(* IEC 61131-3 sources: StarkHacks-Guide-for-PLC-Troubleshooting-Tool/, 8 files *)

(* ---- codesys_constants.st ---- *)
(*
    codesys_constants.st
    Add this as a DUT or global constants list in CODESYS.
    Use these values so the PLC code, Modbus map, Python bridge, and docs all speak the same language.
*)

VAR_GLOBAL CONSTANT
    MODE_IDLE : INT := 0;
    MODE_CONVEYOR : INT := 1;
    MODE_SEQUENCE_TEST : INT := 2;
    MODE_TANK_FILL : INT := 3;
    MODE_HVAC_PUMP : INT := 4;

    FAULT_NONE : INT := 0;
    FAULT_START_BLOCKED_SAFETY : INT := 101;
    FAULT_CONVEYOR_JAM : INT := 201;
    FAULT_SEQUENCE_TIMEOUT : INT := 301;
    FAULT_TANK_FILL_VERIFY : INT := 401;
    FAULT_HVAC_OR_PUMP : INT := 501;
END_VAR

(* ---- codesys_globals.st ---- *)
(*
    codesys_globals.st
    Create a Global Variable List (GVL) in CODESYS and paste this content into it.
    These variables are the shared machine state used by all demo scenarios and the Modbus map.
*)

{attribute 'qualified_only'}
VAR_GLOBAL
    Conveyor_Running : BOOL := FALSE;      (* HR0 *)
    Sensor_Blocked : BOOL := FALSE;        (* HR1 *)
    Motor_Current : INT := 0;              (* HR2 *)
    Safety_OK : BOOL := TRUE;              (* HR3 *)
    Start_Command : BOOL := FALSE;         (* HR4 *)
    Stop_Command : BOOL := FALSE;          (* HR5 *)
    Reset_Command : BOOL := FALSE;         (* HR6 *)
    Tank_Level_Low : BOOL := FALSE;        (* HR7 *)
    Tank_Level_High : BOOL := FALSE;       (* HR8 *)
    Sequence_Timeout : BOOL := FALSE;      (* HR9 *)
    System_Fault_Latch : BOOL := FALSE;    (* HR10 *)
    Pump_Running : BOOL := FALSE;          (* HR11 *)
    HVAC_Fault : BOOL := FALSE;            (* HR12 *)
    Mode_Code : INT := 0;                  (* HR13 *)
    Fault_Code : INT := 0;                 (* HR14 *)

    Demo_EnableAutoCurrentModel : BOOL := TRUE;
    Demo_JamTimerPreset : TIME := T#3S;
    Demo_SequenceTimerPreset : TIME := T#8S;
    Demo_FillGuardPreset : TIME := T#5S;
END_VAR

(* ---- codesys_demo_supervisor.st ---- *)
(*
    codesys_demo_supervisor.st
    Optional helper block for demo stability.
    Call this once per scan to keep unrelated outputs quiet when switching modes.
*)

FUNCTION_BLOCK FB_DemoSupervisor
VAR_INPUT
    Mode_Code : INT;
    Stop_Command : BOOL;
END_VAR
VAR_IN_OUT
    Conveyor_Running : BOOL;
    Pump_Running : BOOL;
END_VAR

IF Stop_Command THEN
    Conveyor_Running := FALSE;
    Pump_Running := FALSE;
END_IF;

CASE Mode_Code OF
    MODE_CONVEYOR, MODE_SEQUENCE_TEST:
        Pump_Running := FALSE;
    MODE_TANK_FILL, MODE_HVAC_PUMP:
        Conveyor_Running := FALSE;
ELSE
    Conveyor_Running := FALSE;
    Pump_Running := FALSE;
END_CASE;

(* ---- codesys_fb_conveyor_demo.st ---- *)
(*
    codesys_fb_conveyor_demo.st
    Function block for conveyor-related demo behavior:
    - start blocked by safety
    - conveyor running logic
    - jam detection
    - sequence timeout support when Mode_Code = 2
*)

FUNCTION_BLOCK FB_ConveyorDemo
VAR_INPUT
    Safety_OK : BOOL;
    Start_Command : BOOL;
    Stop_Command : BOOL;
    Reset_Command : BOOL;
    Sensor_Blocked : BOOL;
    Mode_Code : INT;
    FaultLatchedIn : BOOL;
    JamTimerPreset : TIME;
    SequenceTimerPreset : TIME;
END_VAR
VAR_IN_OUT
    Conveyor_Running : BOOL;
    Motor_Current : INT;
    Sequence_Timeout : BOOL;
    System_Fault_Latch : BOOL;
    Fault_Code : INT;
END_VAR
VAR
    StartEdge : R_TRIG;
    ResetEdge : R_TRIG;
    JamTimer : TON;
    SequenceTimer : TON;
END_VAR

StartEdge(CLK := Start_Command);
ResetEdge(CLK := Reset_Command);

IF Stop_Command THEN
    Conveyor_Running := FALSE;
END_IF;

IF Start_Command AND NOT Safety_OK THEN
    Conveyor_Running := FALSE;
    System_Fault_Latch := TRUE;
    Fault_Code := FAULT_START_BLOCKED_SAFETY;
END_IF;

IF StartEdge.Q AND Safety_OK AND NOT FaultLatchedIn AND (Mode_Code = MODE_CONVEYOR OR Mode_Code = MODE_SEQUENCE_TEST) THEN
    Conveyor_Running := TRUE;
END_IF;

JamTimer(IN := (Mode_Code = MODE_CONVEYOR) AND Conveyor_Running AND Sensor_Blocked, PT := JamTimerPreset);
IF JamTimer.Q THEN
    Conveyor_Running := FALSE;
    System_Fault_Latch := TRUE;
    Fault_Code := FAULT_CONVEYOR_JAM;
END_IF;

SequenceTimer(IN := (Mode_Code = MODE_SEQUENCE_TEST) AND Conveyor_Running AND NOT Sensor_Blocked, PT := SequenceTimerPreset);
IF SequenceTimer.Q THEN
    Sequence_Timeout := TRUE;
    Conveyor_Running := FALSE;
    System_Fault_Latch := TRUE;
    Fault_Code := FAULT_SEQUENCE_TIMEOUT;
END_IF;

IF Conveyor_Running AND Sensor_Blocked THEN
    Motor_Current := 46;
ELSIF Conveyor_Running THEN
    Motor_Current := 18;
ELSE
    Motor_Current := 0;
END_IF;

IF ResetEdge.Q AND Safety_OK AND NOT Sensor_Blocked THEN
    IF Fault_Code = FAULT_CONVEYOR_JAM OR Fault_Code = FAULT_START_BLOCKED_SAFETY OR Fault_Code = FAULT_SEQUENCE_TIMEOUT THEN
        Conveyor_Running := FALSE;
        Sequence_Timeout := FALSE;
        IF Fault_Code <> FAULT_HVAC_OR_PUMP AND Fault_Code <> FAULT_TANK_FILL_VERIFY THEN
            System_Fault_Latch := FALSE;
            Fault_Code := FAULT_NONE;
        END_IF;
    END_IF;
END_IF;

(* ---- codesys_fb_hvac_demo.st ---- *)
(*
    codesys_fb_hvac_demo.st
    Function block for the HVAC / remote pump demo.
*)

FUNCTION_BLOCK FB_HVACDemo
VAR_INPUT
    HVAC_Fault : BOOL;
    Start_Command : BOOL;
    Stop_Command : BOOL;
    Reset_Command : BOOL;
    Mode_Code : INT;
END_VAR
VAR_IN_OUT
    Pump_Running : BOOL;
    System_Fault_Latch : BOOL;
    Fault_Code : INT;
END_VAR
VAR
    ResetEdge : R_TRIG;
END_VAR

ResetEdge(CLK := Reset_Command);

IF Mode_Code <> MODE_HVAC_PUMP THEN
    RETURN;
END_IF;

IF Stop_Command THEN
    Pump_Running := FALSE;
END_IF;

IF Start_Command AND NOT HVAC_Fault AND NOT System_Fault_Latch THEN
    Pump_Running := TRUE;
END_IF;

IF HVAC_Fault THEN
    Pump_Running := FALSE;
    System_Fault_Latch := TRUE;
    Fault_Code := FAULT_HVAC_OR_PUMP;
END_IF;

IF ResetEdge.Q AND NOT HVAC_Fault THEN
    IF Fault_Code = FAULT_HVAC_OR_PUMP THEN
        Pump_Running := FALSE;
        System_Fault_Latch := FALSE;
        Fault_Code := FAULT_NONE;
    END_IF;
END_IF;

(* ---- codesys_fb_tank_fill_demo.st ---- *)
(*
    codesys_fb_tank_fill_demo.st
    Function block for the tank fill verification demo.
*)

FUNCTION_BLOCK FB_TankFillDemo
VAR_INPUT
    Tank_Level_Low : BOOL;
    Tank_Level_High : BOOL;
    Stop_Command : BOOL;
    Reset_Command : BOOL;
    Mode_Code : INT;
    FaultLatchedIn : BOOL;
    FillGuardPreset : TIME;
END_VAR
VAR_IN_OUT
    Pump_Running : BOOL;
    System_Fault_Latch : BOOL;
    Fault_Code : INT;
END_VAR
VAR
    ResetEdge : R_TRIG;
    FillGuardTimer : TON;
END_VAR

ResetEdge(CLK := Reset_Command);

IF Mode_Code <> MODE_TANK_FILL THEN
    FillGuardTimer(IN := FALSE, PT := FillGuardPreset);
    RETURN;
END_IF;

IF Stop_Command THEN
    Pump_Running := FALSE;
END_IF;

IF Tank_Level_Low AND NOT Tank_Level_High AND NOT FaultLatchedIn THEN
    Pump_Running := TRUE;
END_IF;

IF Tank_Level_High THEN
    Pump_Running := FALSE;
END_IF;

FillGuardTimer(IN := Tank_Level_Low AND NOT Tank_Level_High AND NOT Pump_Running, PT := FillGuardPreset);
IF FillGuardTimer.Q THEN
    System_Fault_Latch := TRUE;
    Fault_Code := FAULT_TANK_FILL_VERIFY;
END_IF;

IF ResetEdge.Q AND NOT Tank_Level_Low AND NOT Tank_Level_High THEN
    IF Fault_Code = FAULT_TANK_FILL_VERIFY THEN
        Pump_Running := FALSE;
        System_Fault_Latch := FALSE;
        Fault_Code := FAULT_NONE;
    END_IF;
END_IF;

(* ---- codesys_main_program.st ---- *)
(*
    codesys_main_program.st
    Recommended main PLC program for the demo.

    This version is more modular than plc_logic.st.
    Use this if you want a cleaner CODESYS structure with separate function blocks per scenario.
*)

PROGRAM PLC_PRG
VAR
    ConveyorDemo : FB_ConveyorDemo;
    TankFillDemo : FB_TankFillDemo;
    HVACDemo : FB_HVACDemo;
    DemoSupervisor : FB_DemoSupervisor;
END_VAR

IF GVL_Diagnostics.Reset_Command THEN
    IF GVL_Diagnostics.Safety_OK AND NOT GVL_Diagnostics.Sensor_Blocked AND NOT GVL_Diagnostics.HVAC_Fault THEN
        GVL_Diagnostics.Sequence_Timeout := FALSE;
    END_IF;
END_IF;

DemoSupervisor(
    Mode_Code := GVL_Diagnostics.Mode_Code,
    Stop_Command := GVL_Diagnostics.Stop_Command,
    Conveyor_Running := GVL_Diagnostics.Conveyor_Running,
    Pump_Running := GVL_Diagnostics.Pump_Running
);

ConveyorDemo(
    Safety_OK := GVL_Diagnostics.Safety_OK,
    Start_Command := GVL_Diagnostics.Start_Command,
    Stop_Command := GVL_Diagnostics.Stop_Command,
    Reset_Command := GVL_Diagnostics.Reset_Command,
    Sensor_Blocked := GVL_Diagnostics.Sensor_Blocked,
    Mode_Code := GVL_Diagnostics.Mode_Code,
    FaultLatchedIn := GVL_Diagnostics.System_Fault_Latch,
    JamTimerPreset := GVL_Diagnostics.Demo_JamTimerPreset,
    SequenceTimerPreset := GVL_Diagnostics.Demo_SequenceTimerPreset,
    Conveyor_Running := GVL_Diagnostics.Conveyor_Running,
    Motor_Current := GVL_Diagnostics.Motor_Current,
    Sequence_Timeout := GVL_Diagnostics.Sequence_Timeout,
    System_Fault_Latch := GVL_Diagnostics.System_Fault_Latch,
    Fault_Code := GVL_Diagnostics.Fault_Code
);

TankFillDemo(
    Tank_Level_Low := GVL_Diagnostics.Tank_Level_Low,
    Tank_Level_High := GVL_Diagnostics.Tank_Level_High,
    Stop_Command := GVL_Diagnostics.Stop_Command,
    Reset_Command := GVL_Diagnostics.Reset_Command,
    Mode_Code := GVL_Diagnostics.Mode_Code,
    FaultLatchedIn := GVL_Diagnostics.System_Fault_Latch,
    FillGuardPreset := GVL_Diagnostics.Demo_FillGuardPreset,
    Pump_Running := GVL_Diagnostics.Pump_Running,
    System_Fault_Latch := GVL_Diagnostics.System_Fault_Latch,
    Fault_Code := GVL_Diagnostics.Fault_Code
);

HVACDemo(
    HVAC_Fault := GVL_Diagnostics.HVAC_Fault,
    Start_Command := GVL_Diagnostics.Start_Command,
    Stop_Command := GVL_Diagnostics.Stop_Command,
    Reset_Command := GVL_Diagnostics.Reset_Command,
    Mode_Code := GVL_Diagnostics.Mode_Code,
    Pump_Running := GVL_Diagnostics.Pump_Running,
    System_Fault_Latch := GVL_Diagnostics.System_Fault_Latch,
    Fault_Code := GVL_Diagnostics.Fault_Code
);

(* ---- plc_logic.st ---- *)
(*
    plc_logic.st
    Sample Structured Text logic for the hackathon prototype.

    Notes:
    - Map these variables to the holding registers documented in register_map.md.
    - Factory I/O should drive the simulated sensors and read the actuator outputs.
    - This is a compact demo program, not a production safety program.
*)

PROGRAM PLC_PRG
VAR
    Conveyor_Running : BOOL := FALSE;      (* HR0 *)
    Sensor_Blocked : BOOL := FALSE;        (* HR1 *)
    Motor_Current : INT := 0;              (* HR2 *)
    Safety_OK : BOOL := TRUE;              (* HR3 *)
    Start_Command : BOOL := FALSE;         (* HR4 *)
    Stop_Command : BOOL := FALSE;          (* HR5 *)
    Reset_Command : BOOL := FALSE;         (* HR6 *)
    Tank_Level_Low : BOOL := FALSE;        (* HR7 *)
    Tank_Level_High : BOOL := FALSE;       (* HR8 *)
    Sequence_Timeout : BOOL := FALSE;      (* HR9 *)
    System_Fault_Latch : BOOL := FALSE;    (* HR10 *)
    Pump_Running : BOOL := FALSE;          (* HR11 *)
    HVAC_Fault : BOOL := FALSE;            (* HR12 *)
    Mode_Code : INT := 0;                  (* HR13 *)
    Fault_Code : INT := 0;                 (* HR14 *)

    StartEdge : R_TRIG;
    ResetEdge : R_TRIG;
    JamTimer : TON;
    SequenceTimer : TON;
    FillGuardTimer : TON;
END_VAR

(* Edge detectors *)
StartEdge(CLK := Start_Command);
ResetEdge(CLK := Reset_Command);

(* Defaults *)
Sequence_Timeout := FALSE;

(* Stop command always drops outputs *)
IF Stop_Command THEN
    Conveyor_Running := FALSE;
    Pump_Running := FALSE;
END_IF;

(* Safety blocked start check *)
IF Start_Command AND NOT Safety_OK THEN
    Conveyor_Running := FALSE;
    System_Fault_Latch := TRUE;
    Fault_Code := 101;
END_IF;

(* Healthy start behavior *)
IF StartEdge.Q AND Safety_OK AND NOT System_Fault_Latch THEN
    CASE Mode_Code OF
        1: Conveyor_Running := TRUE;
        2: Conveyor_Running := TRUE;
        3: Pump_Running := Tank_Level_Low AND NOT Tank_Level_High;
        4: Pump_Running := TRUE;
    ELSE
        Conveyor_Running := FALSE;
        Pump_Running := FALSE;
    END_CASE;
END_IF;

(* Conveyor jam logic *)
JamTimer(IN := Conveyor_Running AND Sensor_Blocked, PT := T#3S);
IF JamTimer.Q THEN
    System_Fault_Latch := TRUE;
    Fault_Code := 201;
    Conveyor_Running := FALSE;
END_IF;

(* Sequence timing validation mode *)
SequenceTimer(IN := (Mode_Code = 2) AND Conveyor_Running AND NOT Tank_Level_High, PT := T#8S);
IF SequenceTimer.Q THEN
    Sequence_Timeout := TRUE;
    System_Fault_Latch := TRUE;
    Fault_Code := 301;
    Conveyor_Running := FALSE;
END_IF;

(* Tank fill verification mode *)
IF Mode_Code = 3 THEN
    IF Tank_Level_Low AND NOT System_Fault_Latch THEN
        Pump_Running := TRUE;
    END_IF;

    IF Tank_Level_High THEN
        Pump_Running := FALSE;
    END_IF;

    FillGuardTimer(IN := Tank_Level_Low AND NOT Tank_Level_High AND NOT Pump_Running, PT := T#5S);
    IF FillGuardTimer.Q THEN
        System_Fault_Latch := TRUE;
        Fault_Code := 401;
    END_IF;
END_IF;

(* HVAC / remote pump demo mode *)
IF Mode_Code = 4 THEN
    IF HVAC_Fault THEN
        System_Fault_Latch := TRUE;
        Fault_Code := 501;
        Pump_Running := FALSE;
    END_IF;
END_IF;

(* Motor current model for simulation/diagnostics *)
IF Conveyor_Running AND Sensor_Blocked THEN
    Motor_Current := 46;
ELSIF Conveyor_Running THEN
    Motor_Current := 18;
ELSE
    Motor_Current := 0;
END_IF;

(* Reset logic clears only after fault cause is healthy *)
IF ResetEdge.Q THEN
    IF Safety_OK AND NOT Sensor_Blocked AND NOT HVAC_Fault THEN
        System_Fault_Latch := FALSE;
        Sequence_Timeout := FALSE;
        Fault_Code := 0;
        Conveyor_Running := FALSE;
        IF Mode_Code <> 4 THEN
            Pump_Running := FALSE;
        END_IF;
    END_IF;
END_IF;
